Omron CX-Programmer project 新規ﾌﾟﾛｼﾞｪｸﾄ (CX-Programmer 9.61)

# PLC hoge1: CP1L L

## Program 新規ﾌﾟﾛｸﾞﾗﾑ1 (cyclic task 0)
Local symbols
I 0.00 BOOL
Q 100.00 BOOL

### Section ｾｸｼｮﾝ1

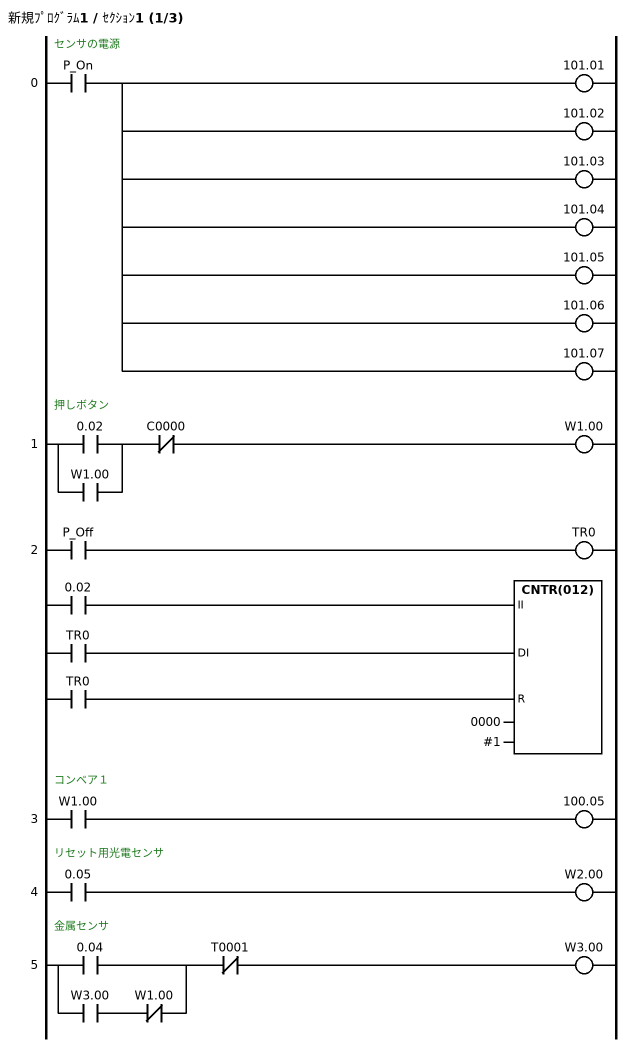
; rung 0: センサの電源
LD P_On
OUT 101.01
OUT 101.02
OUT 101.03
OUT 101.04
OUT 101.05
OUT 101.06
OUT 101.07
; rung 1: 押しボタン
LD 0.02
OR W1.00
ANDNOT C0000
OUT W1.00
; rung 2
LD 0.02
LD P_Off
OUT TR0
LD TR0
CNTR(012) 0000 #1
; rung 3: コンベア１
LD W1.00
OUT 100.05
; rung 4: リセット用光電センサ
LD 0.05
OUT W2.00
; rung 5: 金属センサ
LD 0.04
LD W3.00
ANDNOT W1.00
ORLD
ANDNOT T0001
OUT W3.00

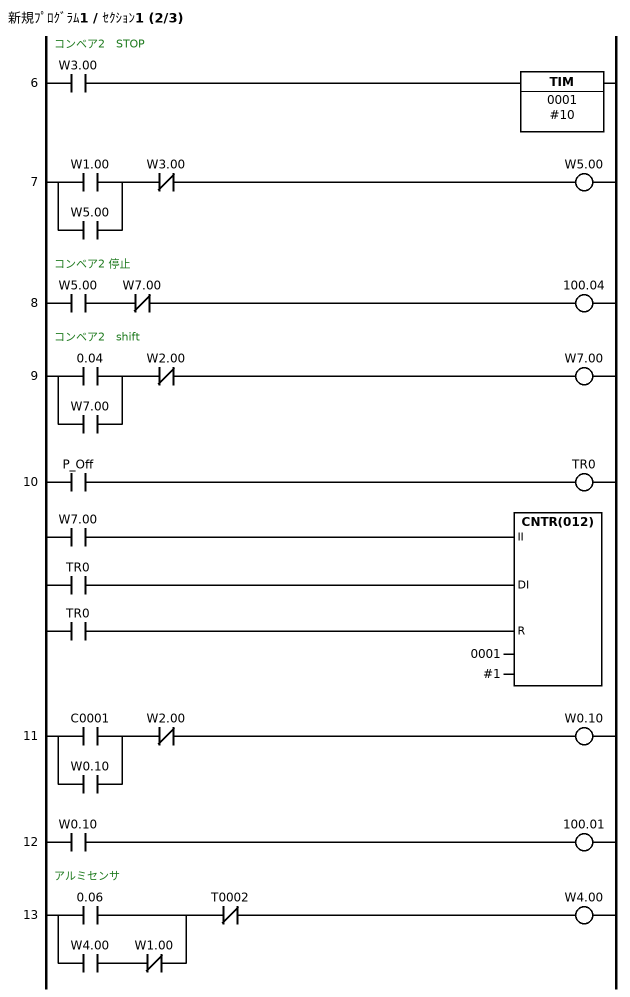
; rung 6: コンベア2　STOP
LD W3.00
TIM 0001 #10
; rung 7
LD W1.00
OR W5.00
ANDNOT W3.00
OUT W5.00
; rung 8: コンベア2 停止
LD W5.00
ANDNOT W7.00
OUT 100.04
; rung 9: コンベア2　shift
LD 0.04
OR W7.00
ANDNOT W2.00
OUT W7.00
; rung 10
LD W7.00
LD P_Off
OUT TR0
LD TR0
CNTR(012) 0001 #1
; rung 11
LD C0001
OR W0.10
ANDNOT W2.00
OUT W0.10
; rung 12
LD W0.10
OUT 100.01
; rung 13: アルミセンサ
LD 0.06
LD W4.00
ANDNOT W1.00
ORLD
ANDNOT T0002
OUT W4.00

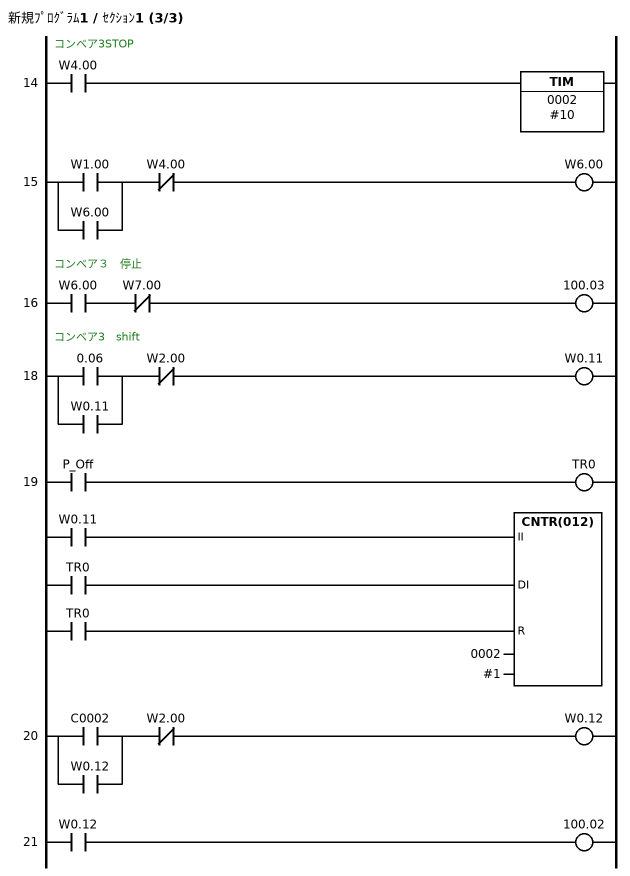
; rung 14: コンベア3STOP
LD W4.00
TIM 0002 #10
; rung 15
LD W1.00
OR W6.00
ANDNOT W4.00
OUT W6.00
; rung 16: コンベア３　停止
LD W6.00
ANDNOT W7.00
OUT 100.03
; rung 18: コンベア3　shift
LD 0.06
OR W0.11
ANDNOT W2.00
OUT W0.11
; rung 19
LD W0.11
LD P_Off
OUT TR0
LD TR0
CNTR(012) 0002 #1
; rung 20
LD C0002
OR W0.12
ANDNOT W2.00
OUT W0.12
; rung 21
LD W0.12
OUT 100.02

### Section END
; rung 0
END(001)